TYPE ASCF_CL_EnumSourceTypes :
STRUCT
	Constante	: INT		:= -1;		//Type: Constant
	None		: INT		:= 0;		//Type: None
	Input		: INT		:= 1;		//Type: Input
	Logic		: INT		:= 2;		//Type: Logic
	Output		: INT		:= 3;		//Type: Output
END_STRUCT
END_TYPE

(* stored: Version 1.1.0.1, ProductVersion 3.1.4026.4
   DUT ASCF_CL_EnumSourceTypes: Id {a8f41747-d0b4-42f1-bc5e-faceb34e3c4d} *)
